// TIA Portal V20 export
TYPE "LAxisCtrl_typeGeneralSettings"
TITLE = LAxisCtrl_typeGeneralSettings
// Support: tech.team.motioncontrol@siemens.com 
// Fax: +49 (0) 9131/98-1297
   STRUCT
      stopOnError : Bool := TRUE;   // TRUE: In case of error the axis will be stopped automatically with fastStop dynamics
      resetWithRestart : Bool := FALSE;   // TRUE: Reinitialization of the technology object and acknowledgment of pending technology alarms. The technology object is reinitialized with the configured start values; FALSE: Acknowledgment of queued technology alarms
      abortWaitingSyncCmd : Bool := TRUE;   // TRUE: Abort waiting synchronous command in case of new basic motion command automatically
   END_STRUCT;
END_TYPE
